FUNCTION_BLOCK TAGIN (* Local Publication of Remote Multicast Data *)
  (* Standard: 61499-1; Function: Communication; Type: Tagged Data *)
  (* Version 0.3, 2007-09-12, JHC, Holobloc Inc, Corrected QO documentation. *)
  (* Version 0.2, 2007-01-13, JHC, Holobloc Inc, Removed CHANNEL, TYPE initializers. *)
  (* Version 0.1, 2006-12-25, JHC, Holobloc Inc, Set QI initial value := 1 *)
  (* Version 0.0, 2006-12-22, JHC, Holobloc Inc, Derived from TAGOUT. *)
  (* Compiler header: package fb.rt.net; *)
  (* Compiler classdef: public class TAGIN extends TAGIO *)
  (* Compiler Java Sun JDK 1.5.0 *)
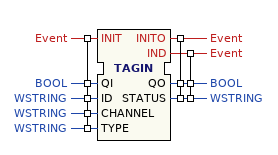
  EVENT_INPUT
    INIT WITH QI, ID, CHANNEL, TYPE; (* Initialization Request *)
  END_EVENT
  EVENT_OUTPUT
    INITO WITH QO, STATUS; (* Initialization Confirm *)
    IND WITH QO, STATUS; (* Communication Status Indication *)
  END_EVENT
  VAR_INPUT
    QI : BOOL := 1; (* 1=Initialize; 0=Terminate *)
    ID : WSTRING; (* Local Multicast Data ID (Default = FB Instance Name) *)
    CHANNEL : WSTRING; (* Remote Subscribe Channel ID *)
    TYPE : WSTRING; (* Comma-separated Tag Datatype List, coerces SUB.RD_x & PUB.SD_x *)
  END_VAR
  VAR_OUTPUT
    QO : BOOL; (* 1=Normal Comms, 0=Comms Error or Termination *)
    STATUS : WSTRING; (* Comms Status *)
  END_VAR
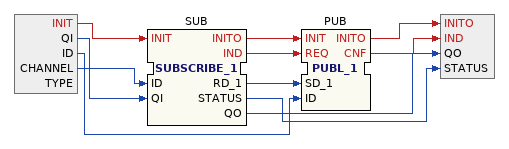
  FBS
    SUB : SUBSCRIBE_1;
    PUB : PUBL_1;
  END_FBS
  EVENT_CONNECTIONS
    INIT TO SUB.INIT;
    SUB.INITO TO PUB.INIT;
    PUB.INITO TO INITO;
    SUB.IND TO PUB.REQ;
    PUB.CNF TO IND;
  END_CONNECTIONS
  DATA_CONNECTIONS
    SUB.RD_1 TO PUB.SD_1;
    CHANNEL TO SUB.ID;
    SUB.STATUS TO STATUS;
    SUB.QO TO QO;
    QI TO SUB.QI;
    ID TO PUB.ID;
  END_CONNECTIONS
END_FUNCTION_BLOCK
